FUNCTION_BLOCK StateMachineBase //IMPLEMENTS  iStateMachine
VAR_INPUT
	resourceID:INT;
END_VAR
VAR_OUTPUT
	//Current alarm code
		//Alarms
	Alarms: ARRAY [0..10] OF BOOL;
	InfoMsg: STRING;
END_VAR
VAR
	//State Machine
	prevState : eState;
	curState : eState;
	nextState : eState;
    HMIState : INT;
	
	cellState : eCellState;
    sTmpState : STRING(255);
    arrStateHistory : ARRAY [ 0..50 ] OF STRING(255);
END_VAR

METHOD abort : BOOL
VAR_INPUT
END_VAR
END_METHOD

METHOD getID : INT
getID:=resourceID;
END_METHOD

METHOD getState : eState
getState:=curState;
END_METHOD

METHOD hold : BOOL
hold := FALSE;
END_METHOD

METHOD ready : BOOL
VAR_INPUT
END_VAR
ready := TRUE;
END_METHOD

METHOD reset : BOOL
reset := FALSE;
END_METHOD

METHOD resetAlarms
VAR_INPUT
END_VAR
VAR
	i:INT;
	ToolData: INT;
END_VAR
FOR i:=1 TO 20 DO
	Alarms[i] := FALSE;
END_FOR
END_METHOD

METHOD resetInfoMsg
VAR_INPUT
END_VAR
InfoMsg := '';
END_METHOD

METHOD restart : BOOL
restart := FALSE;
END_METHOD

METHOD start : BOOL
start := FALSE;
END_METHOD

ACTION StateTransition:
IF curState = eState_error THEN
	resetAlarms();
END_IF

prevState := curState;
curState := nextState;
HMIState := CurState;


sTmpState := TO_STRING(nextState);
Queue_FIFO(
    inputSize   := SIZEOF(sTmpState),
    inputAdr    := ADR(sTmpState),
    arrSize := SIZEOF(arrStateHistory),
    arrAdr  := ADR(arrStateHistory)
);
END_ACTION

METHOD stop : BOOL
stop := FALSE;
END_METHOD

METHOD trackStateChange
VAR_INPUT
END_VAR
END_METHOD

END_FUNCTION_BLOCK

(* stored: Version 1.1.0.1, ProductVersion 3.1.4024.9
   POU StateMachineBase: Id {54cb8061-a005-4e2b-86b3-0c0ca4515e31}, SpecialFunc None
   Method abort: Id {96f0a57a-cfb4-44b2-bd37-4cfe3052afad}
   Method getID: Id {c4b1c257-d4a3-4f35-853a-350d368bdb8c}
   Method getState: Id {fb7b1f04-e557-4d70-913a-963996243d38}
   Method hold: Id {fda735ee-5573-49b6-a1dc-e50a89abc1e6}
   Method ready: Id {ffeb8452-7bbc-4900-b092-b52199c91232}
   Method reset: Id {aa41757f-64fe-4485-a788-8330d90efc9e}
   Method resetAlarms: Id {dee7393a-14d0-406b-8af1-5eb7c794c2f8}
   Method resetInfoMsg: Id {3e9cf03f-1351-481b-a27e-64f1cdf4515e}
   Method restart: Id {224acb1d-42ce-45a3-ae85-ffe9487eb5d4}
   Method start: Id {04c1c909-c569-4ee2-bd8f-e11cd1b0718e}
   Action StateTransition: Id {88062980-a694-48fc-899f-fcd6b677acfc}
   Method stop: Id {a67fa95d-604d-4e25-b7a9-a04ab145fdff}
   Method trackStateChange: Id {28926f83-8ac5-4c34-b170-ff822c7db757} *)
